PROGRAM main
VAR
	Button_Input AT %IX0.0 : bool;
	Light AT %QX0.0 : bool;
	R_TRIG0 : R_TRIG;
END_VAR

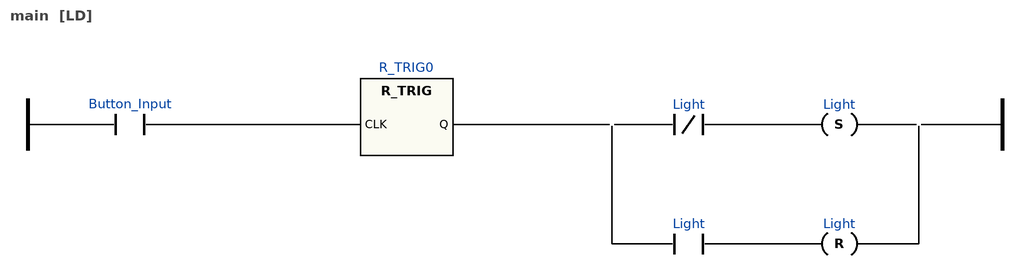
(* LD diagram, written out as Structured Text *)
R_TRIG0(CLK := Button_Input);
IF R_TRIG0.Q AND NOT Light THEN Light := TRUE; END_IF;
IF R_TRIG0.Q AND Light THEN Light := FALSE; END_IF;
END_PROGRAM
